// TIA Portal V17 export
FUNCTION_BLOCK "FB_Motor"   // FB201, LAD
   VAR_INPUT
      Start_Req : Bool;
      Auto_Mode : Bool;
   END_VAR
   VAR_OUTPUT
      Motor_Run : Bool;
   END_VAR
   VAR
      StartDelay : TON_TIME;
   END_VAR
BEGIN

REGION Network 1: Start command interlock
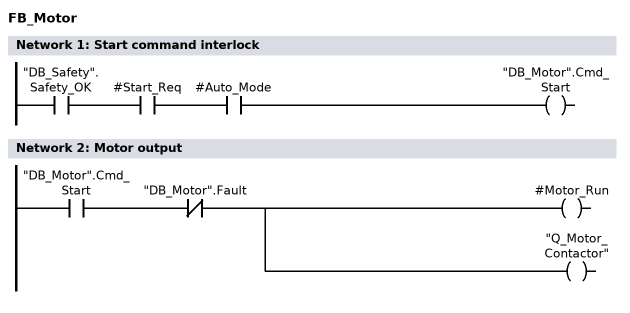
   RUNG wire#powerrail
      Contact( "DB_Safety".Safety_OK )
      Contact( #Start_Req )
      Contact( #Auto_Mode )
      Coil( "DB_Motor".Cmd_Start )
   END_RUNG
   // the same network as SCL:
   "DB_Motor".Cmd_Start := "DB_Safety".Safety_OK AND #Start_Req AND #Auto_Mode;
END_REGION

REGION Network 2: Motor output
   RUNG wire#powerrail
      Contact( "DB_Motor".Cmd_Start )
      I_Contact( "DB_Motor".Fault )
      wire#w1
      Coil( #Motor_Run )
   END_RUNG
   RUNG wire#w1
      Coil( "Q_Motor_Contactor" )
   END_RUNG
   // the same network as SCL:
   #Motor_Run := "DB_Motor".Cmd_Start AND NOT "DB_Motor".Fault;
   "Q_Motor_Contactor" := #Motor_Run;
END_REGION
END_FUNCTION_BLOCK
